(* IEC 61131-3 sources: ae-simplified-sorting-machine/AX/src/stations, 3 files *)

(* ---- BaseStation.st ---- *)
USING System.EdgeDetection;
USING System.Timer;

NAMESPACE SortingMachine
    /// Abstract base class for all station types in the sorting machine
    /// Provides common functionality for enable/disable, state management, error handling, and basic I/O operations
    CLASS ABSTRACT BaseStation
        //=============================================================================
        //SIEMENS AG
        //(c)Copyright 2025 All Rights Reserved
        //-----------------------------------------------------------------------------
        //Tested with:   S7-1500 FW V4.0
        //Engineering:   SIMATIC AX Logic Control Engineering
        //Requirements:  none
        //Functionality: Base class for station control modules in sorting machine
        //-----------------------------------------------------------------------------
        //Change log table:
        //Version  Date       Expert in charge                Changes applied
        //01.00.00 28.11.2025 Siemens Industry Online Support First Release
        //=============================================================================
        VAR PROTECTED
            // Basic control variables
            /// Enable station operation
            _enable : BOOL;
            /// Reset station to initial state
            _reset : BOOL;
            /// Error flag
            _error : BOOL;
            /// Error code
            _status : typeStationStatus := typeStationStatus#STATUS_NO_CALL;

            // Status variables
            /// Station is ready for operation
            _ready : BOOL;
            /// Station is currently processing/moving
            _busy : BOOL;

            // Internal control variables
            /// Rising edge detection for reset
            _resetTrigger : RisingEdge;

            // State machine variables
            /// Current state (0=Idle, 1=Processing, 2=Error)
            _state : typeStationState := typeStationState#STATE_IDLE;
            /// Station Manual mode active
            _manualModeEn : BOOL := FALSE;

            // Station identification
            /// Unique identifier for this station
            _stationID : UINT;
            /// Position of Station in relation to Left reference
            _stationPosLeft : INT;
        END_VAR
        /// Constructor - Initializes the base station with settings
        /// This method should only be used once during startup
        METHOD PROTECTED CONSTRUCTOR
            VAR_INPUT
                /// Unique identifier for this station
                stationID : UINT;
                /// Position of station in relation to left reference
                stationPosLeft : INT;
            END_VAR
            _stationPosLeft := stationPosLeft;
            _stationID := stationID;
            _state := typeStationState#STATE_IDLE;  // Start in idle state
        END_METHOD

        /// Enables the Station for operation
        /// Sets the internal enable flag to allow movement commands
        METHOD PUBLIC Enable // TODO: change variable to public?
            _enable := TRUE;
        END_METHOD

        /// Disables the Station for operation
        /// Sets the internal enable flag to disable movement commands
        METHOD PUBLIC Disable
            _enable := FALSE;
        END_METHOD

        /// Gets the current enable state of the station.
        /// TRUE if station is enabled, FALSE if disabled
        METHOD PUBLIC GetEnable : BOOL
            GetEnable := _enable;
        END_METHOD

        /// Sets the reset signal for the station
        /// Triggers a reset to initial state on rising edge
        METHOD PUBLIC Reset
            _reset := TRUE;
        END_METHOD

        /// Acknowledges errors on the station
        /// Sets the internal acknowledgment flag to clear error conditions
        METHOD PUBLIC AcknowledgeError
            THIS.clearError();
        END_METHOD

        /// Gets the ready status of the station.
        /// TRUE if station is ready for operation, FALSE otherwise
        METHOD PUBLIC GetIsReady : BOOL
            GetIsReady := _ready;
        END_METHOD

        /// Gets the busy/processing status of the station.
        /// TRUE if station is currently processing, FALSE if idle
        METHOD PUBLIC GetIsBusy : BOOL
            GetIsBusy := _busy;
        END_METHOD

        /// Gets the error status of the station.
        /// TRUE if an error has occurred, FALSE if operating normally
        METHOD PUBLIC GetError : BOOL
            GetError := _error;
        END_METHOD

        /// Gets the current error code if an error has occurred.
        METHOD PUBLIC GetStatus : typeStationStatus
            GetStatus := _status;
        END_METHOD

        /// Gets the error code and status of the station using defined type
        METHOD PUBLIC GetErrorAndStatus : typeStatusInterface
            VAR_TEMP
                status : typeStatusInterface;
            END_VAR

            status.error := _error;
            status.status := _status;
            GetErrorAndStatus := status;
        END_METHOD

        /// Gets the current Station ID (UINT) assigned to this station
        METHOD PUBLIC GetStationID : UINT
            GetStationID := _stationID;
        END_METHOD

        /// Set manual mode active state
        METHOD PUBLIC SetManualModeActive
            VAR_INPUT
                /// TRUE to activate manual mode, FALSE to deactivate
                manualModeActvEn : BOOL;
            END_VAR
            _manualModeEn := manualModeActvEn;
        END_METHOD

        /// Sets an error condition with error code
        METHOD PROTECTED setError
            VAR_INPUT
                // Error code to set
                errorCode : typeStationStatus;
            END_VAR
            _error := TRUE;
            _status := errorCode;
            _state := typeStationState#STATE_ERROR_ON; // Go to error state
        END_METHOD

        /// Clears error condition and resets to idle state
        METHOD PROTECTED clearError
            // Reset error feedback variables
            _error := FALSE;
            _status := typeStationStatus#STATUS_NO_CALL;
            // Return to idle state
            _state := typeStationState#STATE_IDLE;
        END_METHOD

        /// Handles common reset functionality.
        /// Should be called by derived classes in their Execute method.
        /// TRUE if reset was triggered this cycle, FALSE otherwise
        METHOD PROTECTED handleReset : BOOL
            // Call trigger for reset so it only works on rising edge
            _resetTrigger(signal := _reset);
            IF _resetTrigger.detected THEN
                _busy := FALSE;
                // Clear errors
                THIS.clearError();
                // Call derived class specific reset
                THIS.onReset();
            END_IF;
            // reset bit for next rising edge detection
            _reset := FALSE;
            // Return value TRUE when trigger was detected
            handleReset := _resetTrigger.detected;
        END_METHOD

        /// Handles common idle state logic
        /// Should be called by derived classes for idle state processing
        METHOD PROTECTED handleIdleState
            _ready := _enable AND NOT _error;
            _busy := FALSE;
        END_METHOD

        /// Handles common error state logic
        /// Should be called by derived classes for error state processing
        METHOD PROTECTED handleErrorState
            _ready := FALSE;
            _busy := FALSE;
            _error := TRUE;
            // Error can only be cleared by reset
        END_METHOD

        /// Abstract method for derived class specific reset operations
        /// Override this method to implement station-specific reset logic
        METHOD PROTECTED ABSTRACT onReset
        END_METHOD

        /// Abstract method for main execution logic
        /// Must be implemented by derived classes
        /// This method should be called cyclically to process station operations
        METHOD PUBLIC ABSTRACT Execute
        END_METHOD
    END_CLASS
END_NAMESPACE

(* ---- ConveyorStationClass.st ---- *)
USING ControlModules;
USING System.EdgeDetection;
USING System.Timer;
USING Simatic.Ax.Sinamics;

NAMESPACE SortingMachine

    /// Conveyor station that manages box transport on a conveyor belt with forward and backward movement.
    /// Handles box addition, removal, and position tracking while preventing collisions between boxes.
    CLASS ConveyorStation EXTENDS BaseStation
        //=============================================================================
        //SIEMENS AG
        //(c)Copyright 2025 All Rights Reserved
        //-----------------------------------------------------------------------------
        //Tested with:   S7-1500 FW V4.0
        //Engineering:   SIMATIC AX Logic Control Engineering
        //Requirements:  none
        //Functionality: Conveyor station class for sorting machine
        //-----------------------------------------------------------------------------
        //Change log table:
        //Version  Date       Expert in charge                Changes applied
        //01.00.00 28.11.2025 Siemens Industry Online Support First Release
        //=============================================================================
        VAR PROTECTED
            // Conveyor specific input variables
            /// Rising edge triggers one step movement
            _move : BOOL;
            /// Add new box at position 0
            _addBox : BOOL;
            /// Data for new box being added
            _newBoxData : BasicBox;

            // Conveyor specific output variables
            /// Conveyor is currently moving
            _moving : BOOL;
            /// Current number of boxes on conveyor
            _boxCount : DINT := DINT#0;
            /// Request to remove the box from conveyor output position
            _readyToRemoveBox : BOOL;
            /// Box was removed and needs to be cleared
            _pendingBoxClear : BOOL := FALSE;

            // Conveyor specific variables
            /// Array of Boxes that should be handled in the call. So the boxes on the Conveyor
            _boxes : ARRAY[BOXES_LOWER_LIMIT..BOXES_UPPER_LIMIT] OF BasicBox;
            /// Size of array 'Boxes'
            _boxesArraySize : DINT := BOXES_UPPER_LIMIT  - BOXES_LOWER_LIMIT + DINT#1 ;

            // Conveyor specific control variables
            /// Rising edge detection for moving conveyor
            _moveTrigger : RisingEdge;
            /// Rising edge detection for add box
            _addBoxTrigger : RisingEdge;
            /// Conveyor control with SinaPos drives
            _conveyorControl : ITransportDevice;

            // Movement control variables
            /// Increment for Moving the boxes to the next position
            _moveIncrement : INT;
            /// Last conveyor position
            _lastConveyorPos : INT := INT#0;
            /// Input Index for next box
            _boxInputIndex  : DINT := DINT#6;
            /// Backward mode enabled
            _conveyorBackwardsEn : BOOL := FALSE;
        END_VAR

        VAR CONSTANT
            BOXES_UPPER_LIMIT : DINT := DINT#6;
            BOXES_LOWER_LIMIT : DINT := DINT#0;
        END_VAR

        /// Constructor - Initializes the conveyor station with control interface and settings
        METHOD PUBLIC CONSTRUCTOR
            VAR_INPUT
                /// Unique identifier for this station
                stationID : UINT;
                /// Position of station in relation to left reference
                stationPosLeft : INT;
                /// Distance increment for each box position movement (default: 128)
                moveIncrement : INT := INT#128;
                /// Interface to the conveyor transport device
                conveyorControl : ITransportDevice;
                /// Index position for new box input (default: BOXES_UPPER_LIMIT)
                boxInputIndex : DINT := BOXES_UPPER_LIMIT;
            END_VAR
            THIS.CONSTRUCTOR(stationID, stationPosLeft);
            _conveyorControl := conveyorControl;
            _moveIncrement := moveIncrement;  // Default move increment
            // Set new input index if within range
            IF boxInputIndex >= BOXES_UPPER_LIMIT THEN
                _boxInputIndex := BOXES_UPPER_LIMIT;
            ELSE
                _boxInputIndex := boxInputIndex;
            END_IF;
        END_METHOD

        /// Set conveyor control interface
        METHOD PUBLIC SetConveyorControl
            VAR_INPUT
                /// Interface to the conveyor transport device
                conveyorControl : ITransportDevice;
            END_VAR
            _conveyorControl := conveyorControl;
        END_METHOD

        /// Implementation of station-specific reset operations.
        /// Clears conveyor-specific data during reset
        METHOD PROTECTED OVERRIDE onReset
            VAR_TEMP
                index : DINT;
            END_VAR
            // Clear all boxes after reset
            FOR index := BOXES_LOWER_LIMIT TO BOXES_UPPER_LIMIT DO
                _boxes[index].ClearData();
            END_FOR;
            _newBoxData.ClearData();
            _boxCount := INT#0;
            _moving := FALSE;
            _move := FALSE;
            _addBox := FALSE;
            _readyToRemoveBox := FALSE;
            _pendingBoxClear := FALSE;
        END_METHOD

        /// Clears error condition and resets to idle state.
        /// Also triggers new box addition in case there is one in line
        METHOD PROTECTED OVERRIDE clearError
            SUPER.clearError();
            // Re-trigger adding box in case box addition was not completed
            _addBox := _newBoxData.BoxData.isPresent;
        END_METHOD

        /// Set manual commands to be done during execute
        METHOD PUBLIC SetManualCommands
            VAR_INPUT
                /// Commands to be executed manually on the elevator
                manualCommands : typeConveyorCommand;
            END_VAR
            // manualCommands.stop is not implemented
            IF manualCommands.moveForward THEN
                THIS.MoveIncrementForward();
            ELSIF manualCommands.moveBackward THEN
                THIS.MoveIncrementBackward();
            END_IF;
        END_METHOD

        /// Sets the add box signal to add a new box at position 0.
        /// TRUE if box prepared to be added to the station. FALSE if rejected
        METHOD PUBLIC AddNewBox : BOOL
            VAR_INPUT
                /// IBasicBox interface containing the box data and triggers adding a new box
                newBox : IBasicBox;
            END_VAR
            IF newBox = NULL THEN
                AddNewBox := FALSE;
                RETURN;
            END_IF;
            // check if possible to add new box, or already waiting to add new box
            IF NOT (_newBoxData.BoxData.isPresent OR _boxes[_boxInputIndex].BoxData.isPresent) THEN
                _newBoxData.CONSTRUCT(newBox.GetBoxData());
                _newBoxData.BoxData.stationNr := _stationID;
                _newBoxData.BoxData.posLeft := _stationPosLeft;
                _addBox := TRUE;
                AddNewBox := TRUE;
            // Deny box addition
            ELSE
                AddNewBox := FALSE;
            END_IF;
        END_METHOD

        /// Checks if the station is ready to remove a box.
        /// TRUE if station has a box ready for removal, FALSE otherwise
        METHOD PUBLIC ReadyToRemoveBox : BOOL
            ReadyToRemoveBox := _readyToRemoveBox;
        END_METHOD

        /// Checks if the station is ready to receive a new box.
        /// Station is ready when no box is present and elevator is at home position.
        /// TRUE if ready to receive a box, FALSE otherwise
        METHOD PUBLIC ReadyToReciveBox : BOOL
            ReadyToReciveBox := NOT (_boxes[_boxInputIndex].BoxData.isPresent OR _moving);
        END_METHOD

        /// Removes the box from the conveyor output position when ready.
        /// Can only remove box when the station indicates it's ready for removal.
        /// Returns the Interface to the removed box, or invalid interface if no box to remove
        METHOD PUBLIC RemoveBox : IBasicBox
            IF _readyToRemoveBox THEN
                RemoveBox := _boxes[BOXES_LOWER_LIMIT];
                _boxCount := _boxCount - 1;
                _pendingBoxClear := TRUE;
                _readyToRemoveBox := FALSE;
            END_IF;
        END_METHOD

        // Conveyor specific property getters
        /// Gets the moving status of the conveyor station
        /// TRUE if conveyor is currently moving, FALSE if stationary
        METHOD PUBLIC GetIsMoving : BOOL
            GetIsMoving := _moving;
        END_METHOD

        /// Initiates an incremental movement operation on the conveyor
        /// Sets the conveyor to moving state to trigger box advancement
        /// This method can be used to manually trigger a single movement step
        METHOD PUBLIC MoveIncrementForward
            IF _boxCount > 0 AND NOT _move THEN
            _conveyorBackwardsEn := FALSE;
            _move := TRUE;
            END_IF;
        END_METHOD

        /// Initiates an incremental movement operation on the conveyor
        /// Sets the conveyor to moving state to trigger box advancement
        /// This method can be used to manually trigger a single movement step
        METHOD PUBLIC MoveIncrementBackward
            IF _boxCount > 0 AND NOT _move THEN
            _conveyorBackwardsEn := TRUE;
            _move := TRUE;
            END_IF;
        END_METHOD

        /// Gets the current number of boxes on the conveyor
        METHOD PUBLIC GetBoxCount : DINT
            GetBoxCount := _boxCount;
        END_METHOD

        /// Gets if the move action is completed
        /// Can be overridden so that other movement methods can be used, like SinaPos
        /// TRUE if move action completed, FALSE if still moving
        METHOD PROTECTED moveDone : BOOL
            moveDone := _conveyorControl.GetIsDone();
        END_METHOD

        METHOD PUBLIC OVERRIDE Enable
            SUPER.Enable();
            _conveyorControl.Enable();
        END_METHOD

        METHOD PUBLIC OVERRIDE Disable
            SUPER.Disable();
            _conveyorControl.Disable();
        END_METHOD

        /// Updates box positions based on conveyor movement
        /// Calculates position delta and moves boxes forward while preventing collisions
        METHOD PROTECTED moveBoxForward
            VAR_TEMP
                deltaPos : INT;
                boxDataFront : typeBoxData;
                boxDataAct : typeBoxData;
                index : DINT;
            END_VAR
            deltaPos := _conveyorControl.GetActualPosition() - _lastConveyorPos;
            // updates all boxes positions. Output box should not move, so start at index 1
            FOR index := BOXES_LOWER_LIMIT + 1 TO _boxInputIndex BY 1 DO
                boxDataAct      := _boxes[index].BoxData;
                // Only continue checking if there is a box in the index
                IF boxDataAct.isPresent THEN
                    boxDataFront    := _boxes[index - 1].BoxData;
                    // Check if move is valid and will not conflict with a box in front of it.
                    // In case there is no box in front, move increment is possible.
                    IF ((boxDataAct.posLeft + deltaPos + boxDataAct.width) <= boxDataFront.posLeft)
                        OR (NOT boxDataFront.isPresent) THEN
                        // Move the box one increment forward
                        _boxes[index].MoveIncrement(deltaPos);
                    END_IF;
                END_IF;
            END_FOR;
            //Update last position
            _lastConveyorPos := _conveyorControl.GetActualPosition();
        END_METHOD

        /// Updates box positions based on conveyor movement
        /// Calculates position delta and moves boxes backwards while preventing collisions
        METHOD PROTECTED moveBoxBackward
            VAR_TEMP
                deltaPos : INT;
                boxDataBack : typeBoxData;
                boxDataAct : typeBoxData;
                index : DINT;
            END_VAR
            deltaPos := _lastConveyorPos - _conveyorControl.GetActualPosition();
            // Updates all boxes positions moving backwards. Start from output box (index 0)
            FOR index := BOXES_LOWER_LIMIT TO (_boxInputIndex - 1) BY 1 DO
                boxDataAct := _boxes[index].BoxData;
                // Only continue checking if there is a box in the index
                IF boxDataAct.isPresent THEN
                    boxDataBack := _boxes[index + 1].BoxData;
                    // Check if move is valid and will not conflict with a box behind it.
                    // In case there is no box behind, move increment is possible.
                    IF ((boxDataAct.posLeft - deltaPos) >= (boxDataBack.posLeft + boxDataBack.width))
                        OR (NOT boxDataBack.isPresent) THEN
                        // Move the box one increment backward
                        _boxes[index].MoveIncrement(- deltaPos);
                    END_IF;
                END_IF;
            END_FOR;
            //Update last position
            _lastConveyorPos := _conveyorControl.GetActualPosition();
        END_METHOD

        /// Main execution method that handles the conveyor station logic
        /// This method should be called cyclically to process conveyor operations
        /// Handles state machine, box movement, error detection, and all conveyor functionality
        METHOD PUBLIC OVERRIDE Execute
            VAR_TEMP
                /// Loop counter
                index : DINT;
            END_VAR
            // Initialize triggers
            _moveTrigger(signal := _move);
            _addBoxTrigger(signal := _addBox);
            // Handle common reset functionality
            THIS.handleReset();
            // Main state machine
            CASE _state OF
                typeStationState#STATE_IDLE: // Idle State
                    THIS.handleIdleState();
                    _moving := FALSE;
                    // Act when station is ready
                    IF _ready THEN
                        // Handle add box request
                        IF _addBoxTrigger.detected  THEN
                            IF _boxCount < _boxesArraySize THEN
                                // Check if last position is free
                                IF NOT _boxes[_boxInputIndex].BoxData.isPresent THEN
                                    // Add new box to the end of the array
                                    _boxes[_boxInputIndex].CONSTRUCT(_newBoxData);
                                    _newBoxData.ClearData(); // Clear newBoxData for next box addition
                                    _boxCount := _boxCount + DINT#1;
                                ELSE
                                    THIS.setError(typeStationStatus#ERR_INPUT_POSITION_OCUPIED); // Add Position occupied
                                END_IF;
                            ELSE
                                THIS.setError(typeStationStatus#ERR_CONV_FULL); // Conveyor full
                            END_IF;
                        END_IF;
                        // Handle step movement request
                        IF _moveTrigger.detected THEN
                            IF  (_boxCount < (_boxInputIndex + 1)) THEN
                                IF _conveyorBackwardsEn THEN
                                    _state := typeStationState#STATE_MOVING_BACKWARD; // Go to moving state
                                    _conveyorControl.PosRelative( - _moveIncrement);
                                    _moving := TRUE;
                                ELSE
                                    _state := typeStationState#STATE_MOVING_FORWARD; // Go to moving state
                                    _conveyorControl.PosRelative(   _moveIncrement);
                                    _moving := TRUE;
                                END_IF;
                            END_IF;
                        END_IF;
                        // Pending clear box
                        IF _pendingBoxClear THEN
                            _boxes[BOXES_LOWER_LIMIT].ClearData();
                            _pendingBoxClear:= FALSE;
                        END_IF;
                        // Check if there's a box at output position and set ready to remove flag
                        IF _boxes[BOXES_LOWER_LIMIT].BoxData.isPresent THEN
                            _readyToRemoveBox := TRUE;
                        END_IF;
                    END_IF;

                typeStationState#STATE_MOVING_FORWARD: // Moving Forward State
                    _moving := TRUE;
                    _ready := FALSE;
                    _busy := TRUE;
                    // Call for Control module control
                    THIS.moveBoxForward();
                    // Wait for movement timer
                    IF THIS.moveDone() THEN
                        // Move all boxes one position forward
                        // Start from the end to avoid overwriting
                        FOR index := BOXES_LOWER_LIMIT TO (_boxInputIndex - 1) BY 1 DO
                            IF _boxes[index + 1].BoxData.isPresent THEN
                                // Check if target position is free
                                IF NOT _boxes[index].BoxData.isPresent THEN
                                    // Move box forward
                                    _boxes[index] := _boxes[index + 1];
                                    // Clear previous position
                                    _boxes[index + 1].ClearData();
                                END_IF;
                            END_IF;
                        END_FOR;
                        _state := typeStationState#STATE_IDLE; // Return to idle state
                    END_IF;

                typeStationState#STATE_MOVING_BACKWARD: // Moving Backward State //TODO: possible to combine with foward?
                    _moving := TRUE;
                    _ready := FALSE;
                    _busy := TRUE;
                    // Call for Control module control
                    THIS.moveBoxBackward();
                    // Wait for movement timer
                    IF THIS.moveDone() THEN
                        // Move all boxes one position backward
                        FOR index := (_boxInputIndex) TO (BOXES_LOWER_LIMIT + 1) BY -1 DO
                            IF _boxes[index - 1].BoxData.isPresent THEN
                                // Check if target position is free. Next entry in case of colision
                                IF _boxes[index].BoxData.isPresent THEN
                                    CONTINUE;
                                END_IF;
                                // Move box backward
                                _boxes[index] := _boxes[index - 1];
                                // Clear previous position
                                _boxes[index - 1].ClearData();
                            END_IF;
                        END_FOR;
                        // Return to idle state
                        _state := typeStationState#STATE_IDLE;
                    END_IF;

                typeStationState#STATE_ERROR_ON: // Error State
                    THIS.handleErrorState();
                    _moving := FALSE;
            END_CASE;
            // Call overwritable call for moving the system
            _conveyorControl.Execute();
            // Reset trigger variables, so that if the variable is not being set, the trigger can be triggered
            THIS.resetTriggers();
        END_METHOD

        /// Resets trigger variables to allow new triggers to be detected
        /// Called at end of execution cycle to clear trigger flags
        METHOD PROTECTED resetTriggers
            _move := FALSE;
            _addBox := FALSE;
        END_METHOD

        /// Get from an array of boxes, all boxes data
        METHOD PUBLIC GetAllBoxData : ARRAY[0.. BOXES_UPPER_LIMIT] OF SortingMachine.typeBoxData
            VAR_TEMP
                /// Temporary Iterator
                index : DINT;
            END_VAR
            FOR index := BOXES_LOWER_LIMIT TO BOXES_UPPER_LIMIT DO
                GetAllBoxData[index] := _boxes[index].BoxData;
            END_FOR;
        END_METHOD

        /// Get from an array of boxes, a box data at specific index.
        METHOD PUBLIC GetBoxDataAtIndex : typeBoxData
            VAR_INPUT
                /// Index of the box to retrieve data from
                index : DINT;
            END_VAR
            GetBoxDataAtIndex := _boxes[index].BoxData;
        END_METHOD

        /// Sets the movement increment value for box positioning
        METHOD PUBLIC SetMoveIncrement
            VAR_INPUT
                /// Distance increment for each box position movement
                increment : INT;
            END_VAR
            _moveIncrement := increment;
        END_METHOD

        /// Gets the current movement increment value
        METHOD PUBLIC GetMoveIncrement : INT
            GetMoveIncrement := _moveIncrement;
        END_METHOD
    END_CLASS
END_NAMESPACE

(* ---- ElevatorBiStateStation.st ---- *)
USING ControlModules;
NAMESPACE SortingMachine
    /// Elevator bi-state station for handling boxes with two-position elevator system
    /// Extends BaseStation to provide elevator-specific functionality for sorting operations
    /// Supports moving boxes to different positions based on box properties
    CLASS ElevatorBiStateStation EXTENDS BaseStation
        //=============================================================================
        //SIEMENS AG
        //(c)Copyright 2025 All Rights Reserved
        //-----------------------------------------------------------------------------
        //Tested with:   S7-1500 FW V4.0
        //Engineering:   SIMATIC AX Logic Control Engineering
        //Requirements:  none
        //Functionality: Elevator bi-state station for sorting machine
        //-----------------------------------------------------------------------------
        //Change log table:
        //Version  Date       Expert in charge                Changes applied
        //01.00.00 28.11.2025 Siemens Industry Online Support First Release
        //=============================================================================
        VAR
            /// Elevator Controller
            _elevatorControl : IElevator;
            /// Calculated position of elevator
            _elevatorPosition : INT ;
            /// Request to remove the boxfrom elevator.
            _readyToRemoveBox : BOOL;
            /// Box was removed and needs to be cleared
            _pendingBoxClear : BOOL := FALSE;
            // Elevator specific variables
            /// Box that should be handled in the call. Elevator can handle only 1 box at a time
            _box : BasicBox;
            /// Station configurations
            _stationConfig : typeElevatorBiStateStationConfig;
        END_VAR

        /// Constructor - Initializes the elevator bi-state station
        METHOD PUBLIC CONSTRUCTOR
            VAR_INPUT
                /// Unique identifier for this station
                stationID : UINT;
                /// Position of station in relation to left reference
                stationPosLeft : INT;
                /// Interface to the elevator control module
                elevatorControl : IElevator;
                /// Configuration parameters for the station
                stationConfig : typeElevatorBiStateStationConfig;
            END_VAR
            THIS.CONSTRUCTOR(stationID, stationPosLeft);
            _elevatorControl := elevatorControl;
            _stationConfig := stationConfig;
        END_METHOD

        /// Set elevator control interface
        METHOD PUBLIC SetElevatorControl
            VAR_INPUT
                /// Interface to the elevator control module
                elevatorControl : IElevator;
            END_VAR
            _elevatorControl := elevatorControl;
        END_METHOD

        /// Gets the box data currently handled by the elevator station
        METHOD PUBLIC GetBoxData : typeBoxData
            GetBoxData := _box.BoxData;
        END_METHOD

        /// Gets the actual position of the elevator
        METHOD PUBLIC GetElevatorPositionValue : INT
            GetElevatorPositionValue := _elevatorPosition;
        END_METHOD

        /// Set manual commands to be done during execute
        /// @param manualCommands: Commands to be executed manually on the elevator
        METHOD PUBLIC SetManualCommands
            VAR_INPUT
                manualCommands : typeElevatorCommand;
            END_VAR
            IF manualCommands.stop THEN
                _elevatorControl.Stop();
            ELSIF manualCommands.moveUp THEN
                _elevatorControl.MoveUp();
            ELSIF manualCommands.moveDown THEN
                _elevatorControl.MoveDown();
            END_IF;
        END_METHOD

        /// Gets the current elevator position as an enumerated value
        /// Converts numeric position to corresponding position enum based on configuration
        METHOD PUBLIC GetElevatorPositionEnum : typeElevatorPosition
            // Determine position based on configured positions
            IF _elevatorPosition = _stationConfig.PositionHome  THEN
                GetElevatorPositionEnum := typeElevatorPosition#HOME;
            ELSIF  _elevatorPosition = _stationConfig.PositionDownLimit THEN
                GetElevatorPositionEnum := typeElevatorPosition#WORK_POS_1;
            ELSIF  _elevatorPosition = _stationConfig.PositionUpLimit THEN
                GetElevatorPositionEnum := typeElevatorPosition#WORK_POS_2;
            ELSE // Unknown position
                GetElevatorPositionEnum := typeElevatorPosition#UNDEF;
            END_IF;
        END_METHOD

        /// Try to add a new box to the elevator. A box can only be added when the elevator is at the right position
        /// and it is free.
        /// TRUE if box added to the station. FALSE if rejected
        METHOD PUBLIC AddNewBox : BOOL
            VAR_INPUT
                /// Interface to the new box to be added
                newBox : IBasicBox;
            END_VAR
            IF newBox = NULL THEN
                AddNewBox := FALSE;
                RETURN;
            END_IF;
            // check if possible to add new box, or already waiting to add new box
            IF NOT THIS.ReadyToReciveBox() THEN
                AddNewBox := FALSE;
                RETURN;
            END_IF;
            // Add the box
            _box.CONSTRUCT(newBox.GetBoxData());
            _box.BoxData.stationNr := (_stationID);
            _box.BoxData.posLeft := (_stationPosLeft);
            AddNewBox := TRUE;
        END_METHOD

        /// Checks if the station is ready to receive a new box.
        /// Box can only be added when elevator is at home position and no box is present.
        /// TRUE if station is ready to remove the box, FALSE otherwise
        METHOD PUBLIC ReadyToRemoveBox : BOOL
            ReadyToRemoveBox := _readyToRemoveBox;
        END_METHOD

        /// Removes the box from the elevator station when ready
        /// Can only remove box when the station indicates it's ready for removal
        /// Returns the Interface to the removed box, or invalid interface if no box to remove
        METHOD PUBLIC RemoveBox : IBasicBox
            IF _readyToRemoveBox THEN
                RemoveBox := (_box);
                _readyToRemoveBox := FALSE;
                _pendingBoxClear := TRUE;
            END_IF;
        END_METHOD

        /// Checks if the station is ready to receive a new box.
        /// Station is ready when no box is present and elevator is at home position.
        /// TRUE if ready to receive a box, FALSE otherwise
        METHOD PUBLIC ReadyToReciveBox : BOOL
            ReadyToReciveBox := NOT _box.BoxData.isPresent AND (_elevatorPosition = _stationConfig.PositionHome);
        END_METHOD

        /// Implementation of station-specific reset operations
        /// Acknowledges any elevator control errors during reset
        METHOD PROTECTED OVERRIDE onReset
            _elevatorControl.AckError();
            _box.ClearData();
            _state := typeStationState#STATE_IDLE;
            _readyToRemoveBox := FALSE;
        END_METHOD

        /// Clears error condition for both station and elevator control
        /// Extends base class error clearing to include elevator control acknowledgment
        METHOD PROTECTED OVERRIDE clearError
            SUPER.clearError();
            _elevatorControl.AckError();
        END_METHOD

        /// Determines target position based on box properties and station configuration.
        /// Uses box base color to determine if elevator should move up, down, or to home.
        /// Returns target position for the elevator based on box properties
        METHOD PROTECTED getTargetPosition : INT
            VAR_TEMP
                boxData : typeBoxData;
            END_VAR
            boxData := _box.BoxData;
            // When there is no box, go to home position
            IF NOT boxData.isPresent THEN
                getTargetPosition := _stationConfig.PositionHome;
                RETURN;
            END_IF;
            // Determine target position based on box base color
            IF boxData.baseColor = _stationConfig.ConditionUp THEN
                getTargetPosition := _stationConfig.PositionUpLimit;
            ELSIF boxData.baseColor = _stationConfig.ConditionDown THEN
                getTargetPosition := _stationConfig.PositionDownLimit;
            ELSE // Unknown box properties, trigger error
                _error := TRUE;
                _status := typeStationStatus#ERR_UNKWNON_BOX;
                getTargetPosition := INT#0;
            END_IF;

        END_METHOD

        /// Checks if the elevator is at the target position within precision limits.
        /// Uses configured precision offset to determine if position is acceptable.
        /// TRUE if elevator is at target position within tolerance, FALSE otherwise
        METHOD PROTECTED isAtTarget : BOOL
            // Check if the position is within the limits
            IF      (_elevatorPosition) >= (THIS.getTargetPosition() - _stationConfig.PrecisionOffset)
                AND (_elevatorPosition) <= (THIS.getTargetPosition() + _stationConfig.PrecisionOffset)  THEN
                isAtTarget := TRUE;
            ELSE
                isAtTarget := FALSE;
            END_IF;
        END_METHOD

        /// Commands the elevator to move towards the target position
        /// Determines direction based on current vs target position and sends appropriate command
        METHOD PROTECTED moveElevator
            // If already at target, don't move
            IF THIS.isAtTarget() THEN
                RETURN;
            END_IF;
            // Get direction to move
            IF _elevatorPosition < THIS.getTargetPosition() THEN
                _elevatorControl.MoveUp();
            ELSE
                _elevatorControl.MoveDown();
            END_IF;
        END_METHOD

        /// Enables both the station and elevator control for operation
        /// Extends base class enable to include elevator control enabling
        METHOD PUBLIC OVERRIDE Enable
            SUPER.Enable();
            _elevatorControl.Enable();
        END_METHOD

        /// Main execution method for the elevator bi-state station
        /// Handles state machine logic for box processing and elevator movement
        /// States: 0=Idle, 1=Moving, 2=Wait Remove Box, 3=Go to Home, 99=Error
        /// This method should be called cyclically to process station operations
        METHOD PUBLIC OVERRIDE Execute
            // check if station or control module is in error to set state machine to error
            IF _elevatorControl.GetIsError() THEN
                THIS.setError(_elevatorControl.GetStatus());
            END_IF;
            // Handle common reset functionality
            THis.handleReset();
            // Clear the input box when pending
            IF _pendingBoxClear THEN
                // Clear all box data
                _box.ClearData();
                _pendingBoxClear := FALSE;
            END_IF;
            // Main state machine
            CASE _state OF
                typeStationState#STATE_IDLE: // Idle State
                    THIS.handleIdleState();
                    // Handle when ready
                    IF _ready AND NOT _manualModeEn THEN
                        // Handle step movement request
                        IF _box.BoxData.isPresent THEN
                            _state := typeStationState#STATE_MOVE_TO_TARGET_POS; // Go to moving state
                        END_IF;
                        // Handle go to Home position after Error or manual mode
                        // with no boxes.
                        IF NOT THIS.isAtTarget() THEN
                            _state := typeStationState#STATE_GO_TO_POS_FOR_NEW_BOX;
                        END_IF;
                    END_IF;

                typeStationState#STATE_MOVE_TO_TARGET_POS: // Moving State
                    _ready := FALSE;
                    _busy := TRUE;
                    // Call for Control module control
                    THIS.moveElevator();
                    // Wait for movement timer
                    IF THIS.isAtTarget() THEN
                        _state := typeStationState#STATE_WAIT_REMOVE_BOX; // Go to removing box state
                        _readyToRemoveBox := TRUE;
                    END_IF;

                typeStationState#STATE_WAIT_REMOVE_BOX:  // Wait Remove Box
                    _ready := FALSE;
                    _busy := TRUE;
                    // When box is removed
                    IF NOT _readyToRemoveBox THEN
                        // Go to home position to be able to accept new boxes
                        _state := typeStationState#STATE_GO_TO_POS_FOR_NEW_BOX;
                    END_IF;

                typeStationState#STATE_GO_TO_POS_FOR_NEW_BOX: // Go to Position to accept new boxes
                    _ready := FALSE;
                    _busy := TRUE;
                    // Call for Control module control
                    THIS.moveElevator();
                    // When Elevator is at the target position
                    IF THIS.isAtTarget() THEN
                        // Go to idle state to wait for further commands
                        _state := typeStationState#STATE_IDLE;
                    END_IF;

                typeStationState#STATE_ERROR_ON: // Error State
                    THIS.handleErrorState();
            END_CASE;
            // Execute call from controller for main logic
            _elevatorControl.Execute();
            // Get position from controller
            _elevatorPosition := _elevatorControl.GetActualPosition();
        END_METHOD
    END_CLASS
END_NAMESPACE
